PROGRAM MAIN
VAR
	Autoritenuta1: FBAutoritenuta;
	Autoritenuta2: FBAutoritenuta;
END_VAR

// prima istanza della auto ritenuta (MSF n.1)
Autoritenuta1(start:= InputOutput.pStart, stop:= InputOutput.pStop, Q => InputOutput.H1);

// seconda istanza della auto ritenuta (MSF n.2)
Autoritenuta2(start:= InputOutput.pStart2, stop:= InputOutput.pStop2 , Q => InputOutput.H2);

END_PROGRAM

(* stored: Version 1.1.0.1, ProductVersion 3.1.4024.12
   POU MAIN: Id {00882d38-10b9-4e7d-9c0c-20e6cbafcfb4}, SpecialFunc None *)
